GLOBALCONSTANTS DefaultPool (* Global constants *)
  PACKAGE Uebungen::const::UT;
  VAR_GLOBAL CONSTANT
    ISO_DESIGNATOR_WIDTH : UINT := 80;
    ISO_DESIGNATOR_HEIGHT : UINT := 80;
    ISO_MASK_SIZE : UINT := 480;
    ISO_VERSION_LABEL : STRING;
    MASK_WIDTH : UINT := 480;
    MASK_HEIGHT : UINT := 480;
    WorkingSet : UINT := 0;
    Macro_Go_To_DataMask_M1 : UINT := 1;
    Macro_Go_To_DataMask_M2 : UINT := 2;
    Macro_Go_To_DataMask_M3 : UINT := 3;
    DataMask_M1 : UINT := 1000;
    Container_B : UINT := 3000;
    Container_low : UINT := 3001;
    Container_medium : UINT := 3002;
    Container_high : UINT := 3003;
    SoftKeyMask_S1 : UINT := 4000;
    SoftKey_F1 : UINT := 5000;
    Button_A1 : UINT := 6000;
    Button_A2 : UINT := 6001;
    Button_A3 : UINT := 6003;
    InputNumber_I3 : UINT := 9002;
    InputNumber_I4 : UINT := 9003;
    OutputString_WorkingSet_0 : UINT := 11000;
    OutputString_SoftKey_F1 : UINT := 11001;
    OutputString_DataMask_M1 : UINT := 11013;
    OutputString_DataMask_M2 : UINT := 11014;
    OutputString_Go_To_DataMask_M1 : UINT := 11015;
    OutputString_Go_To_DataMask_M2 : UINT := 11016;
    OutputString_Button_A1 : UINT := 11017;
    OutputString_Button_A2 : UINT := 11018;
    OutputString_Go_To_DataMask_M3 : UINT := 11026;
    OutputString_Button_A3 : UINT := 11027;
    OutputString_InputNumber_I3 : UINT := 11028;
    OutputString_InputNumber_I4 : UINT := 11029;
    OutputString_OutputNumber_N3 : UINT := 11030;
    OutputNumber_N3 : UINT := 12002;
    Line_W : UINT := 13000;
    Line_S : UINT := 13001;
    Rectangle_black : UINT := 14000;
    Rectangle_grey : UINT := 14001;
    Rectangle_yellow : UINT := 14002;
    Rectangle_red : UINT := 14003;
    information : UINT := 20001;
    alert : UINT := 20002;
    Caution : UINT := 20003;
    Meisterschulen_LogoG1_256 : UINT := 20004;
    Logos_icon : UINT := 20500;
    FontAttributes_6x8 : UINT := 23000;
    FontAttributes_8x12 : UINT := 23001;
    FontAttributes_12x16 : UINT := 23002;
    LineAttributes_black : UINT := 24000;
    LineAttributes_black_3 : UINT := 24001;
    LineAttributes_grey_3 : UINT := 24002;
    LineAttributes_yellow_3 : UINT := 24003;
    LineAttributes_red_3 : UINT := 24004;
    FillAttributes_white : UINT := 25000;
    AuxFunction2_X1 : UINT := 31000;
  END_VAR
END_GLOBALCONSTANTS
